RoboDK station: RunningUR.rdk

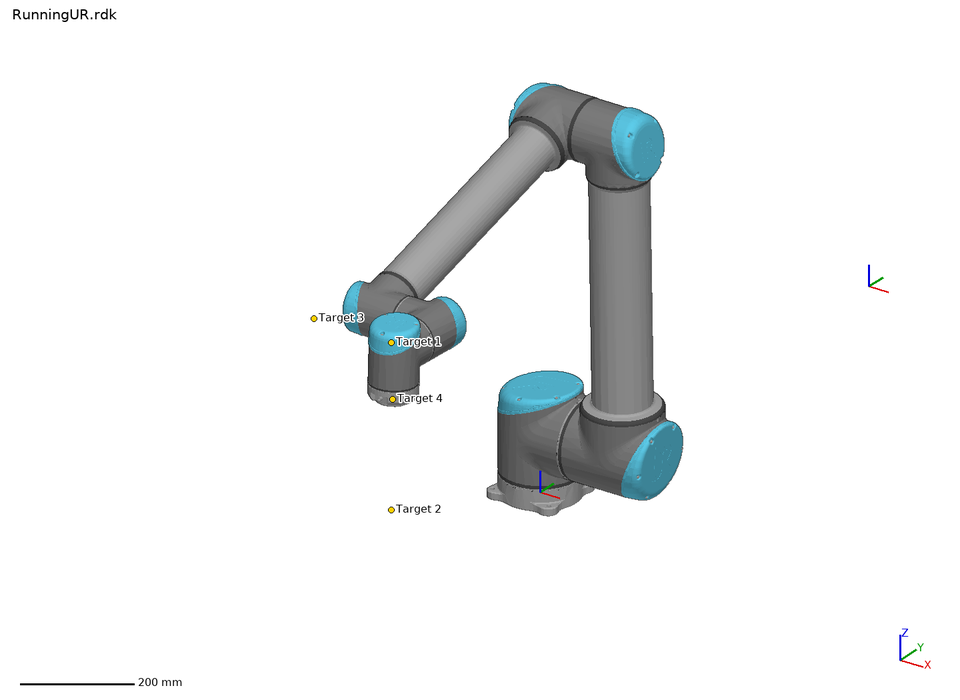
[picture v0: the station drawn from its stored meshes, robots at their saved joint values, targets as dots, program paths as lines]
Station RunningUR (saved by RoboDK 5.9.0). Poses are relative to the parent item; angles as X-Y-Z fixed-axis rotations.
Station parameters (name, value as stored): LIN64
  - frame UR10 Base at (0, 0, 0) mm
    - robot UR10: 6 axes, payload 10 kg, reach 1300 mm, repeatability 0.1 mm, weight 28.9 kg
        modified DH rows (alpha deg, a mm, theta deg, d mm): 0, 0, 0, 128; 90, 0, 180, 0; 0, 612.7, 0, 0; 0, 571.6, 0, 163.9; -90, 0, 0, 115.7; 90, 0, 180, 92.2
        joint limits [-360, -360, -360, -360, -360, -360] to [360, 360, 360, 360, 360, 360]; home [0, -90, -90, 0, 90, 0]; saved at [90.092, -88.631, 104.106, -107.474, -90.17, 1.919]
    - frame Reference_Frame at (0, 1000, 0) mm
      - target Target 1 (Cartesian target) at (163.85, -1687.54, 610.76) mm, rotated rx -179.92 ry 0 rz 179.99 deg; joints [89.996, -89.873, 93.674, -93.881, -90.001, 0.003] of UR10
      - target Target 2 (Cartesian target) at (163.84, -1687.99, 285.47) mm, rotated rx -179.92 ry 0 rz 179.99 deg; joints [89.995, -78.601, 116.498, -127.976, -90.001, 0.002] of UR10
      - target Target 3 (Cartesian target) at (-0.37, -1687.52, 610.77) mm, rotated rx -179.92 ry 0 rz 179.99 deg; joints [76.175, -91.73, 95.502, -93.85, -89.982, -13.818] of UR10
      - target Target 4 (Cartesian target) at (164.73, -1684.1, 499.91) mm, rotated rx -178 ry -0.1 rz 178.17 deg; joints [90.092, -88.631, 104.106, -107.474, -90.17, 1.919] of UR10
